(* LS Electric XG5000 project: 06_Practice_Questions *)
(* PLC LSPLC *)
(* module base 0 slot 0: 입력 모듈:XGI-D21A (DC 24V 입력, 8점 (전류소스/싱크입력)) *)
(* module base 0 slot 1: 출력 모듈:XGQ-RY1A (릴레이 출력, 8점 (2A용, 단독 COM.)) *)

PROGRAM NewProgram (* task: 스캔 프로그램 *)
VAR
    CV : INT;
    Flipflop : FF;
    Flipflop1 : FF;
    P2 AT %IX0.0.2 : BOOL;
    P3 AT %IX0.0.3 : BOOL;
    곱셈결과 : INT;
    곱셈결과2 : UDINT;
    리셋 : BOOL;
    메모리0 AT %MX0 : BOOL;
    모드변환 : BOOL;
    시간 : TIME;
    시간_중간 : UDINT;
    시작 : BOOL;
    업카운터 : CTD_INT;
    업카운터1 : CTU_INT;
    오프타이머1 : TOF;
    오프타이머2 : TOF;
    온타이머1 : TON;
    온타이머2 : TON;
    온타이머3 : TON;
    온타이머4 : TON;
    온타이머5 : TON;
    천 : INT := 1000;
    출력1 : BOOL;
    출력2 : BOOL;
    출력3 : BOOL;
    출력4 : BOOL;
    카운터 : CTU_INT;
    카운터1 : CTU_INT;
    카운트 : INT;
    타이머1 : TP;
    타이머2 : TP;
    타이머3 : TP;
    플립플랍 : FF;
END_VAR

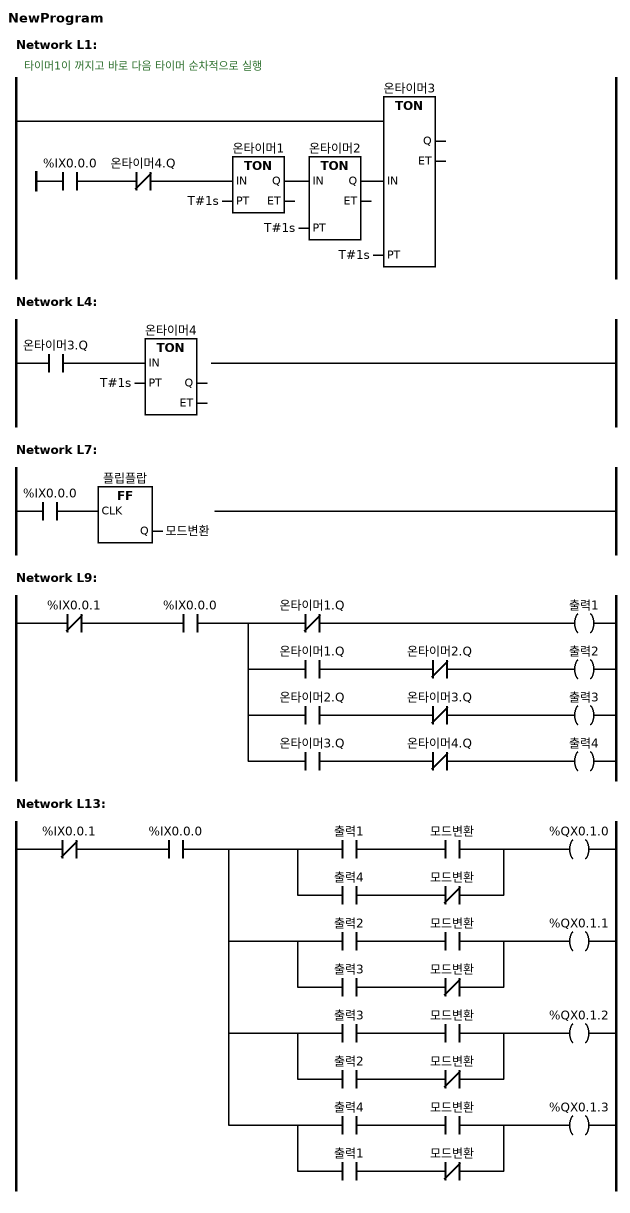
(* 타이머1이 꺼지고 바로 다음 타이머 순차적으로 실행 *)
(* Rung L1 *)
온타이머1(IN := %IX0.0.0 AND NOT 온타이머4.Q, PT := T#1s);
온타이머2(IN := 온타이머1.Q, PT := T#1s);
온타이머3(IN := 온타이머2.Q, PT := T#1s);
(* Rung L4 *)
온타이머4(IN := 온타이머3.Q, PT := T#1s);
(* Rung L7 *)
플립플랍(CLK := %IX0.0.0, Q => 모드변환);
(* Rung L9 *)
출력1 := NOT %IX0.0.1 AND %IX0.0.0 AND NOT 온타이머1.Q;
출력2 := NOT %IX0.0.1 AND %IX0.0.0 AND 온타이머1.Q AND NOT 온타이머2.Q;
출력3 := NOT %IX0.0.1 AND %IX0.0.0 AND 온타이머2.Q AND NOT 온타이머3.Q;
출력4 := NOT %IX0.0.1 AND %IX0.0.0 AND 온타이머3.Q AND NOT 온타이머4.Q;
(* Rung L13 *)
%QX0.1.0 := NOT %IX0.0.1 AND %IX0.0.0 AND ((출력1 AND 모드변환) OR (출력4 AND NOT 모드변환));
%QX0.1.1 := NOT %IX0.0.1 AND %IX0.0.0 AND ((출력2 AND 모드변환) OR (출력3 AND NOT 모드변환));
%QX0.1.2 := NOT %IX0.0.1 AND %IX0.0.0 AND ((출력3 AND 모드변환) OR (출력2 AND NOT 모드변환));
%QX0.1.3 := NOT %IX0.0.1 AND %IX0.0.0 AND ((출력4 AND 모드변환) OR (출력1 AND NOT 모드변환));
END_PROGRAM